FUNCTION_BLOCK ENERGY_COSTS
  {SET_ATTRIBUTE(OpcUa, SERVICE)}
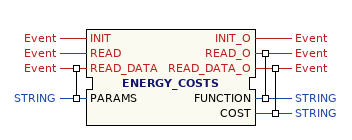
  EVENT_INPUT
    INIT;
    READ;
    READ_DATA WITH PARAMS;
  END_EVENT
  EVENT_OUTPUT
    INIT_O;
    READ_O WITH FUNCTION;
    READ_DATA_O WITH COST;
  END_EVENT
  VAR_INPUT
    PARAMS : STRING; {SET_ATTRIBUTE(OpcUa, Variable)}
  END_VAR
  VAR_OUTPUT
    FUNCTION : STRING; {SET_ATTRIBUTE(OpcUa, Variable)}
    COST : STRING; {SET_ATTRIBUTE(OpcUa, Variable)}
  END_VAR
END_FUNCTION_BLOCK
